{attribute 'reflection'} 
{attribute 'no_explicit_call' := 'do not call this POU directly'} 
FUNCTION_BLOCK FB_VAC_VALVE IMPLEMENTS I_VAC_VALVE
VAR_INPUT
END_VAR
VAR_OUTPUT
END_VAR
VAR
	{attribute 'instance-path'} 
    {attribute 'noinit'} 
	strInstancePath: STRING;
	strFullObjectPath: STRING;
	stEvent: ST_EVENT;
	bAck: BOOL;
	itfOpMode:			I_OP_MODE;
	itfValveVac: I_BASE_VALVE;
	itfSensorVacDetect: I_BINARY_SWITCH;

	
END_VAR

METHOD FB_init : BOOL
VAR_INPUT
	bInitRetains : BOOL; // if TRUE, the retain variables are initialized (warm start / cold start)
	bInCopyCode : BOOL;  // if TRUE, the instance afterwards gets moved into the copy code (online change)
	itfOpMode:	I_OP_MODE;
	itfValveVac: I_BASE_VALVE;
	itfSensorVacDetect: I_BINARY_SWITCH;
END_VAR
THIS^.itfOpMode:= itfOpMode;
THIS^.itfValveVac:= itfValveVac;
THIS^.itfSensorVacDetect:= itfSensorVacDetect;
END_METHOD

{warning 'Methodenimplementierung hinzufügen'}
METHOD M_AllOff
THIS^.itfValveVac.M_Close();
END_METHOD

{warning 'Methodenimplementierung hinzufügen'}
METHOD M_Blow
THIS^.itfValveVac.M_Close();
END_METHOD

{warning 'Methodenimplementierung hinzufügen'}
(*=== Method: M_Run  ============================================

 @brief: Here is the global code (Timer, Event, Flange,...)*)
METHOD M_Run
F_HandleInheritanceObjectInMRun(itfInheritanceObject:=THIS^.itfSensorVacDetect,itfThisObject:=THIS^);
F_HandleInheritanceObjectInMRun(itfInheritanceObject:=THIS^.itfValveVac,itfThisObject:=THIS^);
END_METHOD

{warning 'Methodenimplementierung hinzufügen'}
METHOD M_Vac
THIS^.itfValveVac.M_OPEN();
END_METHOD


(*=== Property: P_Event  ============================================

 @param [set]: 	Set the Structure "ST_EVENT" from another Object
 @param [get]: 	Return the Structure "ST_EVENT", it contains the actual 
					event of the Object *)
PROPERTY P_Event : ST_EVENT
GET
P_Event:= stEvent;
END_GET
SET
END_SET
END_PROPERTY


(*=== Property: P_FullObjectPath  ============================================

 @param [set]: 	Set the Object Path (Clear String of Object)
 @param [get]: 	Return the Objectpath *)
PROPERTY P_FullObjectPath : STRING
GET
P_FullObjectPath:= THIS^.strFullObjectPath;
END_GET
SET
THIS^.strFullObjectPath:= P_FullObjectPath;
END_SET
END_PROPERTY


(*=== Property: P_Global_Ack  ============================================

 @param [set]: 	Set the Bit for Ack from another Object
 @param [get]: 	Return the state of Ack Bit*)
PROPERTY P_Global_Ack : BOOL
GET
P_Global_Ack:= THIS^.bAck;
END_GET
SET
THIS^.bAck:=P_Global_Ack;
END_SET
END_PROPERTY


(*=== Property: P_GlobalID  ============================================

 @param [set]: 	-
 @param [get]: 	Return the string of instance path*)
PROPERTY P_GlobalID : STRING
GET
P_GlobalID:= THIS^.strInstancePath;
END_GET
END_PROPERTY


PROPERTY P_STATE : E_PNEU_VAC_VALVE
GET
IF THIS^.itfValveVac.P_IS_OPEN THEN
	P_STATE:=E_PNEU_VAC_VALVE.Vac_ON_NotDetect;
END_IF

IF THIS^.itfValveVac.P_IS_CLOSE THEN
	P_STATE:=E_PNEU_VAC_VALVE.AllOff;
END_IF

IF THIS^.itfSensorVacDetect.P_Active THEN
	 P_STATE:=E_PNEU_VAC_VALVE.VacDetect;
 END_IF
END_GET
END_PROPERTY

END_FUNCTION_BLOCK

(* stored: Version 1.1.0.1, ProductVersion 3.1.4024.12
   POU FB_VAC_VALVE: Id {95c2ac60-4a73-43d5-ad2a-6b2135c3706b}, SpecialFunc None
   Method FB_init: Id {c2bdda84-fe7f-4acd-9b6a-f6777c879b19}
   Method M_AllOff: Id {642bf660-f5fe-4920-b202-ac9b6cf4f896}
   Method M_Blow: Id {97b01c77-b768-4a6e-b076-172200102cdd}
   Method M_Run: Id {19a56b25-3518-48c1-ba54-b9242c4e9073}
   Method M_Vac: Id {0d0574b3-406c-4a35-9202-108cd803cf40}
   Property P_Event: Id {ab02c34b-e0b5-450b-b361-9f44ad81f258}
   Get Get: Id {917a5898-19db-4242-9e36-bdacf6596f60}
   Set Set: Id {1f67d78d-903a-47aa-8d4c-d77fec12ebe4}
   Property P_FullObjectPath: Id {6af7e757-0f3c-43b9-adaf-0c6109fe1ae2}
   Get Get: Id {8771a41a-207d-4df8-8d2a-01e5b3ebbf7b}
   Set Set: Id {241c1d6f-5618-4f3e-8220-d9007863ec98}
   Property P_Global_Ack: Id {b271ad20-cdb2-48d7-a449-2e415d03d7c6}
   Get Get: Id {0bbbb4f7-4c3c-4c54-bb31-b2fab3894c03}
   Set Set: Id {11f0c9d8-9f78-4390-8f5d-8b4f8c14f2d5}
   Property P_GlobalID: Id {127062cf-7a84-4cd0-8444-211fca33e48a}
   Get Get: Id {ac990de0-26de-43ca-ad22-dbb45d061bb8}
   Property P_STATE: Id {6505177b-afa4-42dd-bf77-7b7ba7114cae}
   Get Get: Id {5cef4b0f-8d6b-439c-84aa-af554d0bd7d3} *)
